DATA_BLOCK "Scanner1LoadData"
{ S7_Optimized_Access := 'FALSE' }
VERSION : 0.1
NON_RETAIN
// ATTRIBUTES
// AUTO_NUMBER = False
// BLOCK_NUMBER = 530
// END_ATTRIBUTES
   STRUCT
      "PLC.Station1DMXCode" : Int;
      "PLC.Station1RecipeNo" : Int;
      "PLC.PartTypeID" : String[128];
      Spare : Byte;
      "MES.ErrorCode" : Int;
      "MES.StatusBits" : DInt;
      "MES.Cycle_ID" : DInt;
      "MES.Unit_ParttypeID" : Int;
   END_STRUCT;


BEGIN

END_DATA_BLOCK

